FUNCTION_BLOCK Day
VAR_INPUT
	
END_VAR
VAR_OUTPUT
END_VAR
VAR
END_VAR

END_FUNCTION_BLOCK

(* stored: Version 1.1.0.1, ProductVersion 3.1.4024.12
   POU Day: Id {1b30805a-7895-4c0e-82ff-d0c87ad5a04b}, SpecialFunc None *)
